FUNCTION_BLOCK Sequencer IMPLEMENTS ISequence, IPLCOpenCall, IPlugin, IPLCOpenCommand
VAR
	i_sequence : SequenceType;
	startStep : ENUM;
	forceStart : BOOL;
	forceDone : BOOL;
	forceError : BOOL;	
	baseManager : StepManagerBasic;
END_VAR

METHOD Aborted : BOOL

i_sequence.activeTasks.Aborted();
END_METHOD

{warning 'add method implementation '}
METHOD AbortPreviousCommands : BOOL
VAR_INPUT
	newCommand	: IPLCOpenCommand;
END_VAR
END_METHOD

METHOD PRIVATE checkStatus : BOOL
VAR
	_commandIndex : INT;
	_anyAbort : BOOL;
	_anyBusy : BOOL;
	_anyError : BOOL;
END_VAR

IF NOT i_sequence.statusChecked THEN
	//We cache the is abort so that we have a consistent 
	//	status for the whole state
	i_sequence.isError := i_sequence.activeTasks.isError;
	i_sequence.isAbort := i_sequence.activeTasks.isAbort;
	i_sequence.isDone := i_sequence.activeTasks.isDone;
END_IF
END_METHOD

{warning 'add property implementation'}
PROPERTY Consume : BOOL
GET
END_GET
END_PROPERTY

{attribute 'monitoring' := 'call'}
PROPERTY CurrentStep : ENUM
GET
currentStep := i_sequence.stepHandler.currentStep;
END_GET
END_PROPERTY

METHOD doStep : ENUM
VAR
END_VAR
IF forceStart THEN
	forceStart := FALSE;
	i_sequence.stepHandler._requestStep(startStep);
END_IF

i_sequence.currentStep := i_sequence.stepHandler.currentStep;
//If the current step has changed,
//	Set the flag for onEntry()
IF i_sequence.stepHandler.RequestNumber <> i_sequence.lastRequestNumber THEN
	
	i_sequence.lastRequestNumber := i_sequence.stepHandler.RequestNumber;
	i_sequence.onEntry := TRUE;
	i_sequence.onExit := FALSE;
ELSE
	i_sequence.onEntry := FALSE;	
END_IF

//The start step is used to detect if the 
i_sequence.startStep := i_sequence.currentStep;

//Mark that we haven't checked the status yet, 
//	This is to ensure we don't have inconsitent onCalls
i_sequence.statusChecked := FALSE;
i_sequence.errorHandled := FALSE;

IF i_sequence.onExit THEN
	doStep := SEQUENCE_STEP.NO_STEP;
ELSE		
	//Return the state
	doStep := i_sequence.currentStep;
END_IF
END_METHOD

METHOD Errored : BOOL
VAR_INPUT
	ID	: INT;
END_VAR
i_sequence.activeTasks.Errored(ID);
END_METHOD

{warning 'add property implementation'}
PROPERTY Execute : BOOL
SET
END_SET
END_PROPERTY

METHOD FB_init : BOOL
VAR_INPUT
	bInitRetains : BOOL; // if TRUE, the retain variables are initialized (warm start / cold start)
	bInCopyCode : BOOL;  // if TRUE, the instance afterwards gets moved into the copy code (online change)
	stepHandler : IStepManager;
END_VAR
IF stepHandler = 0 THEN
	i_sequence.stepHandler :=baseManager;
ELSE
	i_sequence.stepHandler := stepHandler;
END_IF
END_METHOD

METHOD Finished : BOOL
i_sequence.activeTasks.Finished();
END_METHOD

PROPERTY isAbort : BOOL
GET
checkStatus();
isAbort := i_sequence.isAbort;
END_GET
END_PROPERTY

PROPERTY isDone : BOOL
GET
checkStatus();
isDone := i_sequence.isDone;
END_GET
END_PROPERTY

PROPERTY isError : BOOL
GET
checkStatus();
isError := i_sequence.isError;
END_GET
END_PROPERTY

METHOD onAbort : BOOL
VAR_INPUT
	nextStep : ENUM;
END_VAR
//Check all of the status to see if we are aborting

IF isAbort THEN

	IF nextStep >= 0 THEN
		LogMessage( 1, 'Step Abort');
		i_sequence.errorHandled := TRUE;
		setNextStep( nextStep );
	END_IF

	onAbort := TRUE;
ELSE
	onAbort := FALSE;		
END_IF
END_METHOD

METHOD onEntry : BOOL
VAR_INPUT
END_VAR

//If the current step has since the doStep
onEntry := i_sequence.onEntry;
END_METHOD

METHOD onError : BOOL
VAR_INPUT
	nextStep : ENUM;	
END_VAR
IF isError THEN
	IF nextStep >= 0 THEN
		LogMessage( 1, 'Step Abort');
		i_sequence.errorHandled := TRUE;
		setNextStep( nextStep );
	END_IF
	onError := TRUE;
ELSE
	onError := FALSE;		
END_IF
END_METHOD

METHOD onExit : BOOL
VAR_INPUT
END_VAR

//If the current step has since the doStep
onExit := i_sequence.onExit;
END_METHOD

METHOD onFailure : BOOL
VAR_INPUT
	nextStep : ENUM;
END_VAR
IF i_sequence.activeTasks.isAbort OR i_sequence.activeTasks.isError THEN
	//On failure will not set the step if a more specific handler already set the step
	IF i_sequence.errorHandled = FALSE AND nextStep >= 0 THEN
		LogMessage( 1, 'Step Failure');
		setNextStep( nextStep );
	END_IF

	onFailure := TRUE;
ELSE
	onFailure := FALSE;		
END_IF
END_METHOD

METHOD onSuccess : BOOL
VAR_INPUT
	nextStep : ENUM;
END_VAR
IF i_sequence.activeTasks.isDone THEN
	IF nextStep >= 0 THEN
		LogMessage( 1, 'Step Success');
		setNextStep( nextStep );
	END_IF
	
	onSuccess := TRUE;
ELSE
	onSuccess := FALSE;		
END_IF
END_METHOD

{warning 'add method implementation '}
METHOD registerGroup : BOOL
VAR_INPUT
	group	: IPLCOpenGroup;
END_VAR
END_METHOD

{warning 'add property implementation'}
PROPERTY Remote : IPLCOpenCall
GET
END_GET
SET
END_SET
END_PROPERTY

METHOD requestStep : BOOL
VAR_INPUT
	nextStep : ENUM;
END_VAR
i_sequence.stepHandler._requestStep(nextStep);
i_sequence.onExit := TRUE;
END_METHOD

METHOD requestStepClear : BOOL
VAR_INPUT
	nextStep : ENUM;
END_VAR
requestStep(nextStep);
i_sequence.activeTasks.resetCommands();
END_METHOD

METHOD Run : BOOL
THIS^();
END_METHOD

METHOD sequenceAbort : BOOL
VAR_INPUT
	ErrorCode : DINT;
	ErrorMessage: STRING;
END_VAR
i_sequence.stepHandler._sequenceError();
i_sequence.activeTasks.resetCommands();
i_sequence.onExit := TRUE;
END_METHOD

METHOD sequenceComplete : BOOL
VAR_INPUT
END_VAR
i_sequence.stepHandler._sequenceComplete();
i_sequence.activeTasks.resetCommands();
i_sequence.onExit := TRUE;
END_METHOD

METHOD sequenceError : BOOL
VAR_INPUT
	ErrorCode : DINT;
	ErrorMessage: STRING;
END_VAR
i_sequence.stepHandler._sequenceError();
i_sequence.activeTasks.resetCommands();
i_sequence.onExit := TRUE;
END_METHOD

METHOD PROTECTED setNextStep
VAR_INPUT
	nextStep : ENUM;
END_VAR
i_sequence.stepHandler._requestStep(nextStep);
END_METHOD

METHOD Start : BOOL
VAR_INPUT
	Command	: IPLCOpenCommand;
END_VAR
VAR
	_commandIndex : INT;
END_VAR
IF i_sequence.activeTasks.Start(Command) = 0 THEN
	//TODO: All out of commands.. Throw an error
	sequenceError( 10000, 'Too Many Commands in 1 step');
	Start :=  FALSE;
ELSE
	Start :=  TRUE;	
END_IF
END_METHOD

METHOD startSequence : BOOL
VAR_INPUT
END_VAR
requestStep(startStep);
END_METHOD

{warning 'add property implementation'}
PROPERTY status : PLCOpenStatusBase
GET
END_GET
END_PROPERTY

END_FUNCTION_BLOCK

(* stored: Version 1.1.0.1, ProductVersion 3.1.4024.12
   POU Sequencer: Id {6cce11bf-bf75-4b96-8542-c7369e25211e}, SpecialFunc None
   Folder API: Id {939f7e8c-9d25-4182-9029-745e8da56e72}
   Folder Decisions: Id {877b3894-7f7e-462b-b8bc-c682c2070163}
   Folder StateControl: Id {6abf5737-70bc-45fb-a397-53c0f97ae526}
   Folder StateTransition: Id {4654304c-709e-4a34-bdc7-0fda0c88f45a}
   Folder internal: Id {e6aa5ed2-3892-4dae-8fd4-cfebc470258a}
   Folder PLCOpenCaller: Id {692cb7d4-90ad-40a3-84ed-e86faabe0e62}
   Folder PLCOpenCommand: Id {fd5ca5cf-6943-410a-b526-e7c52c8742ad}
   Method Aborted: Id {03503dc0-1791-43ea-b488-bf95491a91d2}
   Method AbortPreviousCommands: Id {3e8b5447-d796-4ea8-80c7-2c28a2a20125}
   Method checkStatus: Id {6b7c3f12-8739-4096-9480-9fa604b0d507}
   Property Consume: Id {c686b2b3-bd51-492d-a98c-896ee2fdb4a5}
   Get Get: Id {44efe948-cca5-435a-a933-d58a8a9393a2}
   Property CurrentStep: Id {b7b67642-2d40-4a87-a0bc-1df8b62b202f}
   Get Get: Id {5106b701-efa0-4091-93e9-d0347cc8550a}
   Method doStep: Id {b100a4e3-ede6-467d-8a89-6654bcb8c169}
   Method Errored: Id {d625b5cc-7ecf-4617-9302-d9a3a7aca5f7}
   Property Execute: Id {70b56461-1624-4c81-b1ce-428ab1a7951c}
   Set Set: Id {b2c36421-446f-4102-bef9-982b63dbf2f6}
   Method FB_init: Id {f87966c2-0adb-4c01-87f6-71b336bb9cc0}
   Method Finished: Id {263545ca-8111-417f-aa03-89bc837548e2}
   Property isAbort: Id {dbaf10d5-3866-4d96-b10f-98bd3ccf9a22}
   Get Get: Id {06516dd3-b590-4e87-bf5f-fded754e45e8}
   Property isDone: Id {0abb87b3-c33c-4d5b-bab6-668ee8ff9e26}
   Get Get: Id {0c5d4645-ee28-4cc6-87d7-b772cfb09f31}
   Property isError: Id {45d11189-3838-46ca-97d2-70f9988c183a}
   Get Get: Id {8849948e-45c2-441d-abda-6c306a83e77e}
   Method onAbort: Id {124a7554-7af0-48f3-9c3b-c6fcfb012c1a}
   Method onEntry: Id {d5293258-9127-40f2-8767-4af37daea8dd}
   Method onError: Id {2b381ad0-9511-4a2a-a59b-89ff6fa0eadc}
   Method onExit: Id {f59d2d40-7d9d-447e-9f98-0b5c912393f5}
   Method onFailure: Id {8864cad6-d51a-434b-b76a-3fb1f56e20e0}
   Method onSuccess: Id {2bf2939a-63ed-4f80-94f9-d2fc5becbe2f}
   Method registerGroup: Id {5f406888-2a46-47ae-9726-a29fd96682c8}
   Property Remote: Id {1baaa5db-8663-490c-a646-fa9e05570894}
   Get Get: Id {fcb1f48e-bcf9-4ced-abb1-06b16eacc58a}
   Set Set: Id {31e61a2d-913f-4239-9a66-18b9d961f4c3}
   Method requestStep: Id {b48e0562-c987-4989-8061-de7cf0c6fe2a}
   Method requestStepClear: Id {a486ef5e-3d7c-419f-8255-b0a39dabc8fc}
   Method Run: Id {77a6af61-d3f7-4c0a-b1d9-a63defd9e3b9}
   Method sequenceAbort: Id {cc629ce3-ace3-4ca4-872b-7b49e09a5e57}
   Method sequenceComplete: Id {f1ae842d-4867-4029-a65e-180592997a50}
   Method sequenceError: Id {06555983-6dc8-4375-b176-7e8590c26dcd}
   Method setNextStep: Id {c0c17481-86c4-4051-a78b-3b1ee372be58}
   Method Start: Id {52f1f4d2-13d6-46fb-aa1f-c1affcffbade}
   Method startSequence: Id {3c531c5d-3c1d-4272-888a-ef0a2888f2c8}
   Property status: Id {68363903-1a6b-41ec-a7c2-c1a657dbfcb5}
   Get Get: Id {a24d3272-022a-44f7-9db8-9409d2cc0db6} *)
